(*
:Description: FUNCTION block to control EtherCAT slave device state machine

:Instructions for use: Requires Tc2_EtherCAT Library

Version history:

+-------------+------------+----------------+----------+------------------------------------------+
|Date         | Version    | created under  | Author   | Remark                                   |
+=============+============+================+==========+==========================================+
|2024-12-12   | 1.0.0.0    | 			    | G.P      | Draft					                  |
+-------------+------------+----------------+----------+------------------------------------------+
|			  | 		   | 			    | 		   | Release							      |
+-------------+------------+----------------+----------+------------------------------------------+

*)
FUNCTION_BLOCK FB_SetSlaveState
VAR_INPUT
	sAMSNet		  AT %I*			: AMSNETID; // Linked to EtherCAT master
    nSlaveAddr    AT %I*     		: UINT;	    //  Linked to PortID of slave device
END_VAR
VAR_OUTPUT
END_VAR
VAR
	fbSetECSlaveState				: Tc2_EtherCAT.FB_EcSetSlaveState;
	fbGetECSlaveState				: Tc2_EtherCAT.FB_EcGetSlaveState;
	_nState							: UINT;
    _sNetId       					: T_AmsNetId; // Must have a value
	_CurrentState					: ST_EcSlaveState;
END_VAR

PROPERTY CurrentState : ST_EcSlaveState
GET
CurrentState := _CurrentState;
END_GET
END_PROPERTY

METHOD GetState : BOOL
VAR_INPUT
	tTimeout   						: TIME := T#10S; // Timeout time for ECSetSlaveState FB
END_VAR
GetState := FALSE;
CASE _nState OF
0:
   _sNetID := F_CreateAmsNetId( sAMSNet ); // Convert linked EtherCAT Master AMS address and convert to string format FB's can use.
   _nState := 1;

1:
  
	// Get slave current state so we can check it changed to the requested state
	fbGetECSlaveState(
		sNetId:= _sNetId , 
		nSlaveAddr:= nSlaveAddr, 
		bExecute:= TRUE, 
		tTimeout:= tTimeout);
		_nState := 2; // Goto next state
  
2:  
	fbGetECSlaveState(bExecute := FALSE, state=> _CurrentState ); // Reset the execute flag of get slave state
	// Check get slave state has completed without errors
	IF (NOT fbGetECSlaveState.bBusy) AND (NOT fbGetECSlaveState.bError) THEN
		_nState := 3; // Move on
	END_IF
3:
   // All complete so reset flags
   GetState := TRUE;
   _nState := 0;

100:
   ;                     // Error handling..
END_CASE
END_METHOD

METHOD ResetStateToOp : BOOL
VAR_INPUT
	tTimeout		: TIME := T#10S; // Timeout time for ECSetSlaveState FB
END_VAR
ResetStateToOp := FALSE;
CASE _nState OF
0:
   _sNetID := F_CreateAmsNetId( sAMSNet ); // Convert linked EtherCAT Master AMS address and convert to string format FB's can use.
   _nState := 1;

1:
   // Set the slave to the state requested to goto	
   fbSetECSlaveState(
	sNetId:= _sNetId, 
	nSlaveAddr:= nSlaveAddr, // Linked port  
	bExecute:= TRUE , 
	tTimeout:= tTimeout , 
	reqState:= 1); // State requested to init
    _nState := _nState + 1; // Goto next state
2:
  
  fbSetECSlaveState( bExecute := FALSE); // Reset the execute flag of set slave state
  // Check the set slave state has completed without errors
  IF (NOT fbSetECSlaveState.bBusy) AND (NOT fbSetECSlaveState.bError) THEN
	 // Get slave current state so we can check it changed to the requested state
	 fbGetECSlaveState(
		sNetId:= _sNetId , 
		nSlaveAddr:= nSlaveAddr, 
		bExecute:= TRUE, 
		tTimeout:= tTimeout);
		_nState := 3; // Goto next state
  END_IF
  
  IF fbSetECSlaveState.bError THEN
	  _nState := 100;
  END_IF
  
3:  
	fbGetECSlaveState(bExecute := FALSE, state=> _CurrentState ); // Reset the execute flag of get slave state
	// Check get slave state has completed without errors
	IF (NOT fbGetECSlaveState.bBusy) AND (NOT fbGetECSlaveState.bError) THEN
		_nState := 4; // Move on
	END_IF
	
4:
	// Make sure in correct state
  	IF _CurrentState.deviceState = Tc2_EtherCAT.EC_DEVICE_STATE_INIT THEN
  	   _nState := _nState + 1; // Goto next state
	END_IF;
	
5:
	// Set the slave to the state requested to goto	
   fbSetECSlaveState(
	sNetId:= _sNetId, 
	nSlaveAddr:= nSlaveAddr, // Linked port  
	bExecute:= TRUE , 
	tTimeout:= tTimeout , 
	reqState:= 8); // State requested to OP
    _nState := _nState + 1; // Goto next state
	
6:
	fbSetECSlaveState( bExecute := FALSE); // Reset the execute flag of set slave state
  	// Check the set slave state has completed without errors
  	IF (NOT fbSetECSlaveState.bBusy) AND (NOT fbSetECSlaveState.bError) THEN
		// Get slave current state so we can check it changed to the requested state
	 	fbGetECSlaveState(
			sNetId:= _sNetId , 
			nSlaveAddr:= nSlaveAddr, 
			bExecute:= TRUE, 
			tTimeout:= tTimeout);
			_nState := _nState + 1; // Goto next state
  	END_IF
  
	IF fbSetECSlaveState.bError THEN
		_nState := 100;
  	END_IF
	
7:  
  	fbGetECSlaveState(bExecute := FALSE, state=> _CurrentState ); // Reset the execute flag of get slave state
	// Check get slave state has completed without errors
	IF (NOT fbGetECSlaveState.bBusy) AND (NOT fbGetECSlaveState.bError) THEN
		_nState := _nState + 1; // Goto next state
	END_IF
	
8:
	// Compare requested state with actual state
  	IF _CurrentState.deviceState = Tc2_EtherCAT.EC_DEVICE_STATE_OP THEN
  	    _nState := _nState + 1; // Goto next state
	END_IF;
	
9:
   // All complete so reset flags
   ResetStateToOp := TRUE;
   _nState := 0;

100:
   ;                     // Error handling..
END_CASE
END_METHOD

METHOD SetState : BOOL
VAR_INPUT
	reqState   						: WORD; // Holds the state the device will be set to 1 = Init, 2 = PreOP, 3 =  Bootstrap, 4 = SafeOp, 8 = OP
    tTimeout   						: TIME := T#10S; // Timeout time for ECSetSlaveState FB
END_VAR
SetState := FALSE;
CASE _nState OF
0:
   _sNetID := F_CreateAmsNetId( sAMSNet ); // Convert linked EtherCAT Master AMS address and convert to string format FB's can use.
   _nState := 1;

1:
   // Set the slave to the state requested to goto	
   fbSetECSlaveState(
	sNetId:= _sNetId, 
	nSlaveAddr:= nSlaveAddr, // Linked port  
	bExecute:= TRUE , 
	tTimeout:= tTimeout , 
	reqState:= reqState); // State requested to goto
    _nState := _nState + 1; // Goto next state
2:
  
  fbSetECSlaveState( bExecute := FALSE); // Reset the execute flag of set slave state
  // Check the set slave state has completed without errors
  IF (NOT fbSetECSlaveState.bBusy) AND (NOT fbSetECSlaveState.bError) THEN
	 // Get slave current state so we can check it changed to the requested state
	 fbGetECSlaveState(
		sNetId:= _sNetId , 
		nSlaveAddr:= nSlaveAddr, 
		bExecute:= TRUE, 
		tTimeout:= tTimeout);
		_nState := 3; // Goto next state
  END_IF
  
  IF fbSetECSlaveState.bError THEN
	  _nState := 100;
  END_IF
  
3:  
	fbGetECSlaveState(bExecute := FALSE, state=> _CurrentState ); // Reset the execute flag of get slave state
	// Check get slave state has completed without errors
	IF (NOT fbGetECSlaveState.bBusy) AND (NOT fbGetECSlaveState.bError) THEN
		_nState := 4; // Move on
	END_IF
4:
	// Compare requested state with actual state
	CASE (reqState) OF
		  1:
		  	IF _CurrentState.deviceState = Tc2_EtherCAT.EC_DEVICE_STATE_INIT THEN
		  	    _nState := 5; // Move to completed state
			END_IF;
		  2:
		  	IF _CurrentState.deviceState = Tc2_EtherCAT.EC_DEVICE_STATE_PREOP THEN
		  	    _nState := 5; // Move to completed state
			END_IF;
          4:
		  	IF _CurrentState.deviceState = Tc2_EtherCAT.EC_DEVICE_STATE_SAFEOP THEN
		  	    _nState := 5; // Move to completed state
			END_IF;
		  8:
		  	IF _CurrentState.deviceState = Tc2_EtherCAT.EC_DEVICE_STATE_OP THEN
		  	    _nState := 5; // Move to completed state
			END_IF;
	  END_CASE
5:
   // All complete so reset flags
   SetState := TRUE;
   _nState := 0;

100:
   ;                     // Error handling..
END_CASE
END_METHOD

END_FUNCTION_BLOCK

(* stored: Version 1.1.0.1, ProductVersion 3.1.4024.12
   POU FB_SetSlaveState: Id {aef72ee8-9f50-4680-a371-6ad716b75c87}, SpecialFunc None
   Property CurrentState: Id {e910f97b-d02d-499b-a64c-15775b80d0b6}
   Get Get: Id {3fbf1cbd-aa02-4e7d-a78d-2baad162b125}
   Method GetState: Id {ef692b14-199b-4434-befb-a4a3c2ca5e22}
   Method ResetStateToOp: Id {fa29bbc0-02d2-4203-8a0e-9b75850ff750}
   Method SetState: Id {b8996a41-8ba6-4c9a-a1cc-b41eb4c74abc} *)
